{attribute 'linkalways'} 
{attribute 'no_explicit_call' := 'This FB is a CLASS and must be accessed using methods or properties'}
{attribute 'enable_dynamic_creation'}
FUNCTION_BLOCK FINAL AND_SINT EXTENDS Node
VAR
	in1 : _SINT(0);
	in2 : _SINT(0);
	out : _SINT(0);
END_VAR

METHOD PUBLIC Clone : I_Node
VAR
	pNode : POINTER TO AND_SINT;
END_VAR
pNode := __NEW(AND_SINT);
Clone := pNode^;
END_METHOD

METHOD FB_init : BOOL
VAR_INPUT
	bInitRetains : BOOL; // if TRUE, the retain variables are initialized (warm start / cold start)
	bInCopyCode : BOOL;  // if TRUE, the instance afterwards gets moved into the copy code (online change)
END_VAR
AddInput('in1',THIS^.in1);
AddInput('in2',THIS^.in2);
AddOutput('out', THIS^.out);
END_METHOD

METHOD PROTECTED OnExecute
VAR
END_VAR
out.Value := in1.Value AND in2.Value;
END_METHOD

END_FUNCTION_BLOCK

(* stored: Version 1.1.0.1, ProductVersion 3.1.4024.15
   POU AND_SINT: Id {170ba094-258d-4970-991c-89f2299d7801}, SpecialFunc None
   Folder Constructor: Id {3fbd6277-ebc6-493e-9ee6-e748a25559e1}
   Method Clone: Id {e5f418fd-f4fd-4f3e-87c3-1b6915d47b9f}
   Method FB_init: Id {ed7bed82-a692-4cfa-91e9-1e777c58d78e}
   Method OnExecute: Id {12d1fd95-8873-4344-aa9f-f5c21643b26c} *)
